TYPE VTD_Instruction_DUT :
STRUCT
	Mode_Change:  UINT;
	Stop:  BOOL;
	Enable:  Bool;
	Execulte:  Bool;
	Reset:  Bool;
	Pallet_Type:  UInt;
	Task_ID:  UInt;
	Task_Metadata:  String;
	Move_To_Level:  UInt;
	Manual_Up:  Bool;
	Manual_Down:  Bool;
	Manual_LP_Retract:  Bool;
	Manual_LP_Extend:  Bool;
	Start_Teach:  BOOL;
END_STRUCT
END_TYPE

(* stored: Version 1.1.0.1
   DUT VTD_Instruction_DUT: Id {67e3d87d-f38e-4875-a53d-74adf9aeedcf} *)
